FUNCTION_BLOCK Test_F_PadString_PadsShortStrings EXTENDS T_UnitTestBase
VAR
    SubjectString : T_MaxString;
    ResultString  : T_MaxString;
END_VAR

{attribute 'analysis' := '-33'} // inhibit unused variable warning
METHOD RunTest
IF Retest THEN
	SUPER^.Init();
END_IF

IF TestCompleted THEN
	RETURN;
END_IF

SubjectString := 'Bob';
ResultString  := F_PadString(InputString := SubjectString,
                             Length      := 20);

AssertEquals_INT(Expected := 20,
                 Actual   := LEN(ResultString),
                 Message  := 'LEN(ResultString)');

AssertEquals_STRING(Expected := 'Bob                 ',
                    Actual   := ResultString,
                    Message  := 'ResultString');

TestCompleted := TRUE;
END_METHOD

END_FUNCTION_BLOCK

(* stored: Version 1.1.0.1, ProductVersion 3.1.4024.12
   POU Test_F_PadString_PadsShortStrings: Id {027d78fd-7523-426a-a6c3-d6c4d9f6c3fb}, SpecialFunc None
   Method RunTest: Id {f9993575-954a-060f-16d4-b4076f995ccf} *)
